(* CODESYS project WagoSysSQL_SQLiteExample.ecp

Project tree, tasks and I/O mapping:
  PFC200_G2_4ETH_CAN_USB : 750-8212 PFC200 G2 2ETH RS, WAGO, order no. 0750-8212, version 5.16.3.16
    application Application
      libraries: ; WagoSysSQL_SQLite, 1.0.1.2 (WAGO); WagoTypesSQL_SQLite, 1.0.1.1 (WAGO)
      task DB2_Task (cyclic, interval t#2ms, priority 4) calls DB2_PRG
      task DB_Task (cyclic, interval t#1ms, priority 5) calls DB_PRG
      20 Program Organization Units/
        program DB_PRG [ST]
        function block FbSQLite3 [ST]: Close, Column_Text, Errmsg, FB_exit, FB_init, Finalize, Open, Prepare, Step, Column_Int
        program DB2_PRG [ST]
        function FuByteArrayToString [ST]
        function FuStudentToString [ST]
      29 Types/
        data type Student
      global variables GlobalState
    ProjectConfiguration
    ProjectConfigurationTxt
    Kbus : Kbus, WAGO, version 1.4.0.2
        unmapped channels: K-BUS diagnostics
    MODBUS
      MODBUS : MODBUS, WAGO, order no. n/a, version 1.1.1.16
    Serial
      COM1 : COM1, WAGO, version 0.0.0.19
    Common.PCI
    EtherNet/IP
      Ethernet : Ethernet, WAGO, version 35.16.0.0
  PNIDL_PFC200_G2_4ETH_CAN_USB_GenericMaster : Generic Master, WAGO, order no. None, version 1.0.0.0
    PNIDL_PFC200_G2_4ETH_CAN_USB : 750-8215, WAGO, order no. 750-8215, version SW=, HW=
        settings: Slave parameters.DeviceId = 4846; Slave parameters.Identification.Subnet mask = [255,255,255,0]; Module parameters.Module ident number = 2684354561; DAPInfo.SharedDeviceSupported = True; DAPInfo.DeviceAccessSupported = True; DAPInfo.LLDP_NoD_Supported = True; DAPInfo.CheckDeviceID_Allowed = True; DAPInfo.IOXS_Required = True; DAPInfo.ResetToFactoryModes = 20; DAPInfo.AddressAssignment = 1; DAP Submodule.Submodule ident number = 1; SubmoduleState = 32767; IM1.'Function' = 'Wago.Fieldbus.Profinet.DeviceCore.DataItems.Gsdml.VisibleStringItem'; IM1.'Location' = 'Wago.Fieldbus.Profinet.DeviceCore.DataItems.Gsdml.VisibleStringItem'; 34cc7c09-c9de-4ab8-9d2c-ec632b521310 = '2018-02-28 11:52'; 7dfa2bca-dd55-42c9-8f93-cd5821bfdf60 = 'Wago.Fieldbus.Profinet.DeviceCore.DataItems.IMDescriptorItem'; Xn.Submodule ident number = 4096; Xn.Subslot number = 32768; SubmoduleState = 32767; InterfaceSubmoduleInfo.PTP_BoundarySupported = True; InterfaceSubmoduleInfo.DCP_BoundarySupported = True; InterfaceSubmoduleInfo.StartupModeAdvanced_supp = True; InterfaceSubmoduleInfo.StartupModeLegacy_supp = True; X1.Submodule ident number = 4097; X1.Subslot number = 32769; SubmoduleState = 32767; PortSubmoduleInfo.PortDeactivationSupported = True; PortSubmoduleInfo.CheckMAUTypeSupported = True; X2.Submodule ident number = 4097; X2.Subslot number = 32770; SubmoduleState = 32767; PortSubmoduleInfo.PortDeactivationSupported = True; PortSubmoduleInfo.CheckMAUTypeSupported = True
  PNIDL_PFC200_G2_4ETH_CAN_USB_GenericMaster_1 : Generic Master, WAGO, order no. None, version 1.0.0.0
    PNIDL_PFC200_G2_4ETH_CAN_USB : 750-8215, WAGO, order no. 750-8215, version SW=, HW=
        settings: Slave parameters.DeviceId = 4846; Slave parameters.Identification.Subnet mask = [255,255,255,0]; Module parameters.Module ident number = 2684354561; DAPInfo.SharedDeviceSupported = True; DAPInfo.DeviceAccessSupported = True; DAPInfo.LLDP_NoD_Supported = True; DAPInfo.CheckDeviceID_Allowed = True; DAPInfo.IOXS_Required = True; DAPInfo.ResetToFactoryModes = 20; DAPInfo.AddressAssignment = 1; DAP Submodule.Submodule ident number = 1; SubmoduleState = 32767; IM1.'Function' = 'Wago.Fieldbus.Profinet.DeviceCore.DataItems.Gsdml.VisibleStringItem'; IM1.'Location' = 'Wago.Fieldbus.Profinet.DeviceCore.DataItems.Gsdml.VisibleStringItem'; 05c39bcc-548b-4498-87ca-9cb2675d4560 = '2018-03-05 11:46'; 6911cab9-1290-4d2f-9571-7f12c038e139 = 'Wago.Fieldbus.Profinet.DeviceCore.DataItems.IMDescriptorItem'; Xn.Submodule ident number = 4096; Xn.Subslot number = 32768; SubmoduleState = 32767; InterfaceSubmoduleInfo.PTP_BoundarySupported = True; InterfaceSubmoduleInfo.DCP_BoundarySupported = True; InterfaceSubmoduleInfo.StartupModeAdvanced_supp = True; InterfaceSubmoduleInfo.StartupModeLegacy_supp = True; X1.Submodule ident number = 4097; X1.Subslot number = 32769; SubmoduleState = 32767; PortSubmoduleInfo.PortDeactivationSupported = True; PortSubmoduleInfo.CheckMAUTypeSupported = True; X2.Submodule ident number = 4097; X2.Subslot number = 32770; SubmoduleState = 32767; PortSubmoduleInfo.PortDeactivationSupported = True; PortSubmoduleInfo.CheckMAUTypeSupported = True
  00000000-0000-0000-0000-000000000000|C:\Users\MarkusF\AppData\Local\Temp\2ebcf6317f4145cf9ac5cb2a904c88e7\ProjectCfg.txt
  00000000-0000-0000-0000-000000000000|C:\Users\MarkusF\AppData\Local\Temp\5e58910f149a45f99028891ad1d6cabc\Project.xml
*)

// PFC200_G2_4ETH_CAN_USB/Application/29 Types/Student
TYPE Student :
STRUCT
	Name : STRING;
	Age : STRING;
	City: STRING;
END_STRUCT
END_TYPE

// PFC200_G2_4ETH_CAN_USB/Application/GlobalState
{attribute 'qualified_only'}
VAR_GLOBAL
	xIsSqliteInitialized: BOOL:= FALSE;	
END_VAR

// PFC200_G2_4ETH_CAN_USB/Application/20 Program Organization Units/DB2_PRG
(*
	This program 
 		1. opens the database from the file '/home/db.sqlite'.
		2. enables Write Ahead Log mode in SQLite (readers don't block writers and vice versa)
		3. creates the table 'students' if it does not exit
		4. inserts all students from 'initStudents' into the students table
		5. reads back all students from table students and proceeds with 4.
		
	The database will grow over time up to the point where all diskspace is used.
	
*)

PROGRAM DB2_PRG
VAR	
	database: FbSQLite3('/home/db.sqlite'); // instance of the sqlite wrapper fb 
	state: INT := 0; // the state variable. 
	err : DINT; // error variable, holds the last sqlite3 return value
	
	(* Some data to insert into the database *)
	initStudents : ARRAY[0..3] OF Student := 
		[(Name:= 'Eric', Age:='8', City:= 'Berlin'),
 		(Name:= 'Stan', Age:='8', City:= 'Amsterdam'),
		(Name:= 'Kyle', Age:='9', City:= 'London'),
	    (Name:= 'Kenny', Age:='9', City:= 'Peking')];
						
	counter : INT := 0;    // counter variable, used during insert (does not count to 11)
	currStudent : Student; // holds the current student that is read back from the database
	
	sSql: STRING(255);   // holds the current sql statement	
	sTemp : STRING(255); // temp string, used to create the 'insert student' sql string
	sErrorMsg : STRING;  // holds the last sqlite3 error message in human readable english
END_VAR

(*
	This program 
 		1. opens the database from the file '/home/db.sqlite'.
		2. enables Write Ahead Log mode in SQLite (readers don't block writers and vice versa)
		3. creates the table 'students' if it does not exit
		4. inserts all students from 'initStudents' into the students table
		5. reads back all students from table students and proceeds with 4.
		
	The database will grow over time up to the point where all diskspace is used.
*)


CASE state OF
	0: 
		(* open the database and go to the next state when successfull *)
		err := database.Open();
		IF database.xIsOpen THEN
			state:= 1;
		END_IF
		
	1: 
		(* THIS STEP IS OPTIONAL
		   Demonstrate on how to use the sqlite3 PRAGMA
		   
		   As an example we enable the Write Ahead Log mode of sqlite. Before doing this you
	       should understand the implication this has. 
		*)
		err := database.Prepare('PRAGMA journal_mode=WAL');
		IF err = WagoSysSQL_SQLite.ErrorCodes.gc_SQLITE_OK THEN
			err := database.Step();
		END_IF
		GlobalState.xIsSqliteInitialized := TRUE;
		database.Finalize();
		state := 10;	
	
	10:	
	    (* Create the table 'students' if it does not exist already *)		
		err:= database.Prepare('create table if not exists students (Name TEXT, Age TEXT, City TEXT)');
		IF err = WagoSysSQL_SQLite.ErrorCodes.gc_SQLITE_OK THEN
			(* the statement was prepared, now execute it *)
			err := database.Step();
			IF err = WagoSysSQL_SQLite.ErrorCodes.gc_SQLITE_DONE THEN
				(* the table was created or already existed, proceed with inserting some data in state 20 *)				
				state := 20;
			ELSE
				state := 99;
			END_IF			
		END_IF
		(* finalize the prepared statement *)
		err := database.Finalize();
		
	20:
	    (* in this state we insert all entries from ``initStudents`` into the students table - one row per cycle *)
		
		(* Get a student formatted as string like "Name", "Age", "City" *)
		sTemp := FuStudentToString(initStudents[counter]);
		(* put the string formatted student into the sql statement *)
		sSql := Format1('insert into students values (%s)', ADR(sTemp));
		(* prepare the sql statement *)
		err := database.Prepare(sSql);		
		IF err = WagoSysSQL_SQLite.ErrorCodes.gc_SQLITE_OK THEN
			err := database.Step();			
			IF err = WagoSysSQL_SQLite.ErrorCodes.gc_SQLITE_DONE THEN
				(* when the insert was successfull increase counter by 1 *) 				
				counter := counter + 1;			
			ELSIF err <> WagoSysSQL_SQLite.ErrorCodes.gc_SQLITE_BUSY THEN
				(* something went wrong *) 				
				state := 99;
			END_IF
			
			IF counter >= 4 THEN
				(* all entries from initStudents are inserted go to the next state *)
				counter:= 0;
				state := 30;
			END_IF			
		END_IF
		err := database.Finalize();
		
	30: 
	    (* prepare the select statement to read all students *)
		sSQl := 'select Name, Age, City from students';
		err := database.Prepare(sSql);		
		IF err = WagoSysSQL_SQLite.ErrorCodes.gc_SQLITE_OK THEN
			(* proceed to the next state ``Step()``-ing through result of select*) 
			state := 40;
		ELSE
			(* unhandled retrun code => goto error state *)
			state:= 99;
		END_IF			
		
	40: 
		(* step through the result *)
		err := database.Step();
		IF err = WagoSysSQL_SQLite.ErrorCodes.gc_SQLITE_ROW THEN
			(* we found a row, now extract all the columns *)
			currStudent.Name :=  database.Column_Text(0);
			currStudent.Age :=  database.Column_Text(1);
			currStudent.City :=  database.Column_Text(2);
		ELSIF err = WagoSysSQL_SQLite.ErrorCodes.gc_SQLITE_DONE THEN
			(* we stepped through the result *)
			(* finalize the select statement and proceed with inserting some more students *)  
			database.Finalize();
			state := 20;
			counter := 0;
		ELSE
			(* unhandled retrun code => goto error state *)
			state:= 99;
		END_IF		

	99:	
		(* Aww, Snap!
		   Something went wrong => preserve the error message and close the database.
		   Never again leave this state!
		*) 
		IF err <> WagoSysSQL_SQLite.ErrorCodes.gc_SQLITE_OK THEN
			sErrorMsg := database.Errmsg();
			err := WagoSysSQL_SQLite.ErrorCodes.gc_SQLITE_OK;
			database.Finalize();
			database.Close();
		END_IF
		
END_CASE

IF err <> WagoSysSQL_SQLite.ErrorCodes.gc_SQLITE_OK THEN
	sErrorMsg := database.Errmsg();
END_IF

END_PROGRAM

// PFC200_G2_4ETH_CAN_USB/Application/20 Program Organization Units/FuStudentToString
FUNCTION FuStudentToString : STRING
VAR_INPUT
	student: Student;
END_VAR
VAR
END_VAR

FuStudentToString := Format3('"%s", "%s", "%s"', ADR(student.Name), ADR(student.Age), ADR(student.City));

END_FUNCTION

// PFC200_G2_4ETH_CAN_USB/Application/20 Program Organization Units/FbSQLite3
(*
	Encapsulates the usage of ``WagoSysSQL_SQLite``.
	
	 WagoSysSQL_SQLite should always be encapsulated in some sort of Function Block in order to guarantee
	 that all the resources that sqlite3 allocates are safely deallocated in case of
		- Reset
		- Download
	 
	  ``FbSQLite3`` is an example on how an ecapsulation could look like. In practice you would probably build
	  another Function Block ontop of ``FbSQLite3`` which provides an abstraction of the database operations
	  and hides all the SQL-specific methods.	  
*)

FUNCTION_BLOCK FbSQLite3
VAR_INPUT
END_VAR
VAR_OUTPUT
	xIsOpen: BOOL;
	xIsPrepared: BOOL;
END_VAR
VAR
	sqlite3: WagoSysSQL_SQLite.typSQLite3;
	sqlite3_stmt: WagoSysSQL_SQLite.typSQLite3_Stmt;	
	sFilename: STRING(256);
END_VAR

(*
	Close the Database Connection
*)
METHOD PUBLIC Close : DINT
VAR_INPUT
END_VAR
IF xIsOpen THEN
	(* Finalize the prepared statement, so we don't leak any memory *)
	IF xIsPrepared THEN		
		Finalize();
	END_IF
	(* Close the database *)
	Close := WagoSysSQL_SQLite.FuSqlite3_Close(ADR(sqlite3));
	xIsOpen := FALSE;
END_IF
END_METHOD

(*
	Get the content of the passed column in text format.	
	:note: The result is encoded in UTF8.
*)
METHOD Column_Text: STRING
VAR_INPUT
	diColumn: DINT;	
END_VAR
VAR
	sText: STRING;	
END_VAR
IF xIsOpen AND xIsPrepared THEN
	WagoSysSQL_SQLite.FuSqlite3_Column_Text(ADR(sqlite3_stmt), diColumn, ADR(sText), SIZEOF(sText));
	Column_Text := sText;
END_IF
END_METHOD

(*
	Translates the current error in human readable text (english)
*)
METHOD Errmsg : STRING
VAR_INPUT
END_VAR
VAR
	pBytes : POINTER TO STRING(256);
	sStringBuffer : STRING(256);
	udiActualSize : UDINT;
END_VAR
pBytes := ADR(sStringBuffer);
FuSqlite3_Errmsg(ADR(sqlite3), pBytes, SIZEOF(sStringBuffer), ADR(udiActualSize));
Errmsg := pBytes^;
END_METHOD

(*
	Destructor
	Takes care that all resources allocated by sqlite3 are cleaned up in case of Reset or Program Download.
*)

METHOD FB_exit : BOOL
VAR_INPUT 
 bInCopyCode : BOOL; //  TRUE: The exit method is called in order to leave the instance, which will be copied afterwards (Online-Change). 
END_VAR
(* don't change the state of this instance during online change *)
IF NOT bInCopyCode THEN
	IF xIsPrepared THEN
		Finalize();
	END_IF
	IF xIsOpen THEN
		Close();
	END_IF
END_IF
END_METHOD

(*
	Constructor of the FB.
	Stores the given database filename in a private variable.
*)
METHOD FB_init: BOOL
VAR_INPUT
  bInitRetains : BOOL; // TRUE: the retain variables are initialized (reset warm / reset cold)
  bInCopyCode : BOOL;  // TRUE the instance will be copied to the copy-code afterward (online change)
  sDatabaseFilename: STRING(256); // filename of the database 
END_VAR
sFilename := sDatabaseFilename;
END_METHOD

(*
	Finalize a prepared statement.
*)
METHOD Finalize : DINT
VAR_INPUT
END_VAR
IF xIsPrepared THEN
	Finalize:= WagoSysSQL_SQLite.FuSqlite3_Finalize(ADR(sqlite3_stmt));
	xIsPrepared := FALSE;
END_IF
END_METHOD

(*
	Opens the sqlite database.
*)
METHOD PUBLIC Open : DINT
IF NOT xIsOpen THEN
	Open := WagoSysSQL_SQLite.FuSqlite3_Open(sFilename, ADR(sqlite3));
	xIsOpen := Open = WagoSysSQL_SQLite.ErrorCodes.gc_SQLITE_OK;	
END_IF
END_METHOD

(*
	Prepares the given SQL-statement.
	On success, use ``Step()`` to execute the statement.
	
*)
METHOD Prepare: DINT
VAR_INPUT
	sSql: STRING(512);
END_VAR
IF xIsOpen AND NOT xIsPrepared THEN
	Prepare := WagoSysSQL_SQLite.FuSqlite3_Prepare(ADR(sqlite3), ADR(sSql), ADR(sqlite3_stmt));
	xIsPrepared := Prepare = WagoSysSQL_SQLite.ErrorCodes.gc_SQLITE_OK;
END_IF
END_METHOD

(*
	Executes a ``Prepare()``-ed statement.
*)
METHOD Step : DINT
VAR_INPUT
END_VAR
IF xIsOpen AND xIsPrepared THEN
	Step := WagoSysSQL_SQLite.FuSqlite3_Step(ADR(sqlite3_stmt));
END_IF
END_METHOD

METHOD Column_Int : DINT
VAR_INPUT
	diColumn: DINT;	
END_VAR
IF xIsOpen AND xIsPrepared THEN
	Column_Int := WagoSysSQL_SQLite.FuSqlite3_Column_Int(ADR(sqlite3_stmt), diColumn);	
END_IF
END_METHOD

END_FUNCTION_BLOCK

// PFC200_G2_4ETH_CAN_USB/Application/20 Program Organization Units/DB_PRG
(*
	This program 
 		1. opens the database from the file '/home/db.sqlite'.		
		2. inserts all students from 'initStudents' into the students table
		3. reads back all students from table students and proceeds with 2.
		
	The database will grow over time up to the point where all diskspace is used.
	
*)

PROGRAM DB_PRG
VAR	
	database: FbSQLite3('/home/db.sqlite'); // instance of the sqlite wrapper fb 
	state: INT := 0; // the state variable. 
	err : DINT; // error variable, holds the last sqlite3 return value
	
	(* Some data to insert into the database *)
	initStudents : ARRAY[0..3] OF Student := 
		[(Name:= 'Sharon', Age:='42', City:= 'Tokyo'),
 		(Name:= 'Sheila', Age:='43', City:= 'Barcelona'),
		(Name:= 'Carol', Age:='44', City:= 'Moscow'),
	    (Name:= 'Linda', Age:='45', City:= 'Hong Kong')];
						
	counter : INT := 0;    // counter variable, used during insert (does not count to 11)
	currStudent : Student; // holds the current student that is read back from the database
	
	sSql: STRING(255);   // holds the current sql statement	
	sTemp : STRING(255); // temp string, used to create the 'insert student' sql string
	sErrorMsg : STRING;  // holds the last sqlite3 error message in human readable english
END_VAR

(*
	This program 
 		1. opens the database from the file '/home/db.sqlite'.
		2. enables Write Ahead Log mode in SQLite (readers don't block writers and vice versa)
		3. creates the table 'students' if it does not exit
		4. inserts all students from 'initStudents' into the students table
		5. reads back all students from table students and proceeds with 4.
		
	The database will grow over time up to the point where all diskspace is used.
*)

// Wait for DB2_PRG to initialize the database 
IF NOT GlobalState.xIsSqliteInitialized THEN
	return;
END_IF


CASE state OF
	0: 
		(* open the database and go to the next state when successfull *)
		err := database.Open();
		IF database.xIsOpen THEN
			state:= 20;
		END_IF
		
	20:
	    (* in this state we insert all entries from ``initStudents`` into the students table - one row per cycle *)
		
		(* Get a student formatted as string like "Name", "Age", "City" *)
		sTemp := FuStudentToString(initStudents[counter]);
		(* put the string formatted student into the sql statement *)
		sSql := Format1('insert into students values (%s)', ADR(sTemp));
		(* prepare the sql statement *)
		err := database.Prepare(sSql);		
		IF err = WagoSysSQL_SQLite.ErrorCodes.gc_SQLITE_OK THEN
			err := database.Step();			
			IF err = WagoSysSQL_SQLite.ErrorCodes.gc_SQLITE_DONE THEN
				(* when the insert was successfull increase counter by 1 *) 				
				counter := counter + 1;			
			ELSIF err <> WagoSysSQL_SQLite.ErrorCodes.gc_SQLITE_BUSY THEN
				(* something went wrong *) 				
				state := 99;
			END_IF
			
			IF counter >= 4 THEN
				(* all entries from initStudents are inserted go to the next state *)
				counter:= 0;
				state := 30;
			END_IF			
		END_IF
		err := database.Finalize();
		
	30: 
	    (* prepare the select statement to read all students *)
		sSQl := 'select Name, Age, City from students';
		err := database.Prepare(sSql);		
		IF err = WagoSysSQL_SQLite.ErrorCodes.gc_SQLITE_OK THEN
			(* proceed to the next state ``Step()``-ing through result of select*) 
			state := 40;
		ELSE
			(* unhandled retrun code => goto error state *)
			state:= 99;
		END_IF			
		
	40: 
		(* step through the result *)
		err := database.Step();
		IF err = WagoSysSQL_SQLite.ErrorCodes.gc_SQLITE_ROW THEN
			(* we found a row, now extract all the columns *)
			currStudent.Name :=  database.Column_Text(0);
			currStudent.Age :=  database.Column_Text(1);
			currStudent.City :=  database.Column_Text(2);
		ELSIF err = WagoSysSQL_SQLite.ErrorCodes.gc_SQLITE_DONE THEN
			(* we stepped through the result *)
			(* finalize the select statement and proceed with inserting some more students *)  
			database.Finalize();
			state := 20;
			counter := 0;
		ELSE
			(* unhandled retrun code => goto error state *)
			state:= 99;
		END_IF		

	99:	
		(* Aww, Snap!
		   Something went wrong => preserve the error message and close the database.
		   Never again leave this state!
		*) 
		IF err <> WagoSysSQL_SQLite.ErrorCodes.gc_SQLITE_OK THEN
			sErrorMsg := database.Errmsg();
			err := WagoSysSQL_SQLite.ErrorCodes.gc_SQLITE_OK;
			database.Finalize();
			database.Close();
		END_IF
		
END_CASE

IF err <> WagoSysSQL_SQLite.ErrorCodes.gc_SQLITE_OK THEN
	sErrorMsg := database.Errmsg();
END_IF

END_PROGRAM

// PFC200_G2_4ETH_CAN_USB/Application/20 Program Organization Units/FuByteArrayToString
FUNCTION FuByteArrayToString : STRING
VAR_INPUT
	pbIn: POINTER TO BYTE;
END_VAR
VAR
	psStr : POINTER TO STRING;
END_VAR

psStr := pbIn;
FuByteArrayToString:= psStr^;

END_FUNCTION
